// TIA Portal V18 export
FUNCTION_BLOCK "SafetyGate"   // FB5200, LAD
{ S7_Optimized_Access := 'FALSE' }
// stored: AutoNumber false, SetENOAutomatically false
   VAR_INPUT
      iSysInface : "RCS_SysComInterface_V1";
      "iSafetyGate Opened Monitor" : Bool;   // 安全门打开状态监控
      "iSafetyGate Locked Monitor" : Bool;   // 安全门锁定状态监控
      i1s_Pulse : Bool;   // 1s脉冲信号
      "iSafetyGate AutoLock Timer" : Time := T#1s;   // 安全门自动模式下锁延时
      "iSafetyGate ManualLock Timer" : Time := T#60s;   // 安全门手动模式下锁定延时
      iMode : Int;
   END_VAR
   VAR_OUTPUT
      "oSafetyGate LockedLamp" { ExternalAccessible := 'False'; ExternalVisible := 'False'; ExternalWritable := 'False'} : Bool;   // 安全门解锁输出状态
   END_VAR
   VAR_IN_OUT
      ioSafetyGateLock : Bool;   // 安全门锁定输出
      ioHMI_Interface : "SafetyGateUDT";
   END_VAR
   VAR
      "sSafetyGate Timer" { S7_SetPoint := 'True'} : Array[1..5] of TON_TIME;
      sP_Trig : Array[1..10] of Bool;
      sN_Trig : Array[1..10] of Bool;
      "sSafetyGate UnlockRequest" { ExternalAccessible := 'False'; ExternalVisible := 'False'; ExternalWritable := 'False'} : Bool;   // 安全门开门请求标志位
      "sSafetyGate LockRequest" : Bool;
   END_VAR
   VAR_TEMP
      tAlyways_On : Bool;
      tAlyways_Off : Bool;
   END_VAR
   VAR_TEMP   // added for the SCL form of the ladder/FBD networks
      _w1 : Bool;
      _w2 : Bool;
      _w3 : Bool;
      _w4 : Bool;
      _w5 : Bool;
   END_VAR
BEGIN

REGION Network 1: #tAlyways_On
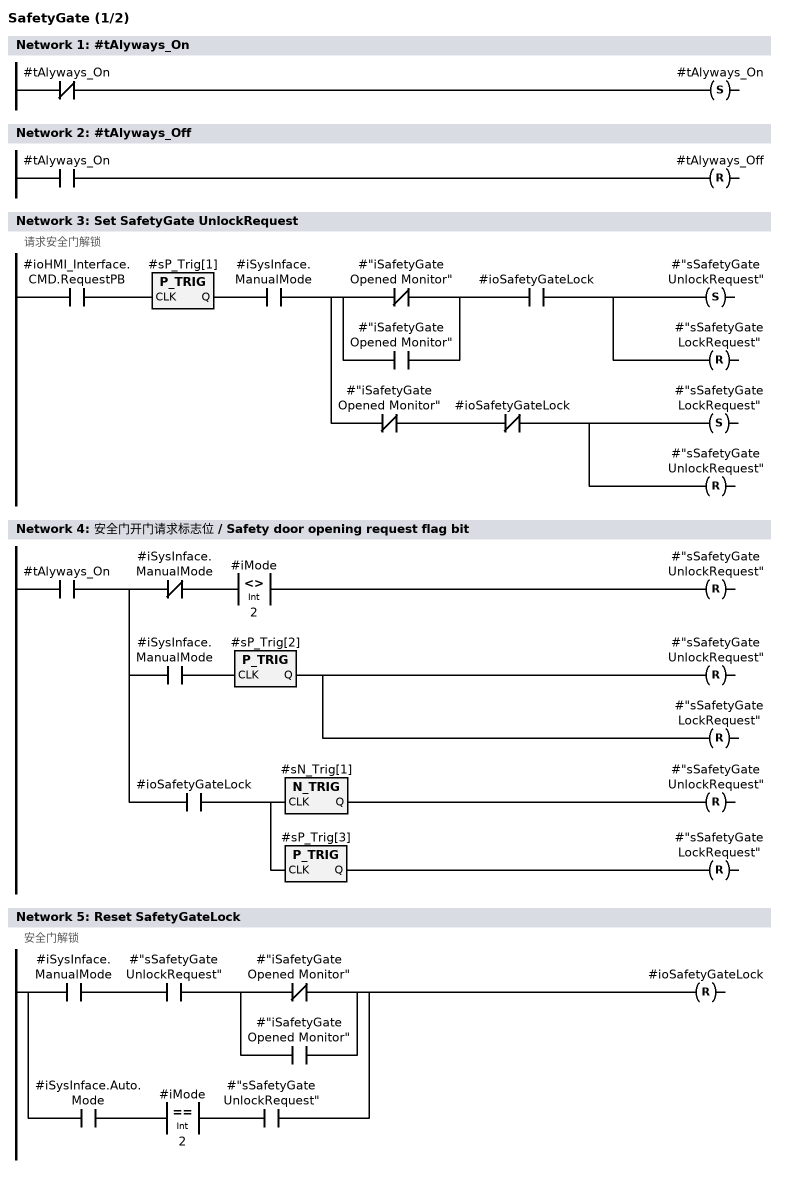
   RUNG wire#powerrail
      I_Contact( #tAlyways_On )
      S_Coil( #tAlyways_On )
   END_RUNG
   // the same network as SCL:
   IF NOT #tAlyways_On THEN #tAlyways_On := TRUE; END_IF;
END_REGION

REGION Network 2: #tAlyways_Off
   RUNG wire#powerrail
      Contact( #tAlyways_On )
      R_Coil( #tAlyways_Off )
   END_RUNG
   // the same network as SCL:
   IF #tAlyways_On THEN #tAlyways_Off := FALSE; END_IF;
END_REGION

REGION Network 3: Set SafetyGate UnlockRequest
   // 请求安全门解锁
   RUNG wire#powerrail
      Contact( #ioHMI_Interface.CMD.RequestPB )
      P_Trig( #sP_Trig[1] )
      Contact( #iSysInface.ManualMode )
      wire#w1
      I_Contact( #"iSafetyGate Opened Monitor" )
      wire#w2
      Contact( #ioSafetyGateLock )
      wire#w3
      S_Coil( #"sSafetyGate UnlockRequest" )
   END_RUNG
   RUNG wire#w1
      Contact( #"iSafetyGate Opened Monitor" )
   END_RUNG wire#w2
   RUNG wire#w3
      R_Coil( #"sSafetyGate LockRequest" )
   END_RUNG
   RUNG wire#w1
      I_Contact( #"iSafetyGate Opened Monitor" )
      I_Contact( #ioSafetyGateLock )
      wire#w4
      S_Coil( #"sSafetyGate LockRequest" )
   END_RUNG
   RUNG wire#w4
      R_Coil( #"sSafetyGate UnlockRequest" )
   END_RUNG
   // the same network as SCL:
   #_w1 := #ioHMI_Interface.CMD.RequestPB AND NOT #sP_Trig[1];   // rising edge
   #sP_Trig[1] := #ioHMI_Interface.CMD.RequestPB;
   #_w2 := #_w1 AND #iSysInface.ManualMode;
   IF #_w2 AND (NOT #"iSafetyGate Opened Monitor" OR #"iSafetyGate Opened Monitor") AND #ioSafetyGateLock THEN
       #"sSafetyGate UnlockRequest" := TRUE;
       #"sSafetyGate LockRequest" := FALSE;
   END_IF;
   IF #_w2 AND NOT #"iSafetyGate Opened Monitor" AND NOT #ioSafetyGateLock THEN
       #"sSafetyGate LockRequest" := TRUE;
       #"sSafetyGate UnlockRequest" := FALSE;
   END_IF;
END_REGION

REGION Network 4: 安全门开门请求标志位 / Safety door opening request flag bit
   RUNG wire#powerrail
      Contact( #tAlyways_On )
      wire#w1
      I_Contact( #iSysInface.ManualMode )
      { S7_Templates := "SrcType := Int" } NE_Contact(in1 := #iMode, in2 := 2)
      R_Coil( #"sSafetyGate UnlockRequest" )
   END_RUNG
   RUNG wire#w1
      Contact( #iSysInface.ManualMode )
      P_Trig( #sP_Trig[2] )
      wire#w2
      R_Coil( #"sSafetyGate UnlockRequest" )
   END_RUNG
   RUNG wire#w2
      R_Coil( #"sSafetyGate LockRequest" )
   END_RUNG
   RUNG wire#w1
      Contact( #ioSafetyGateLock )
      wire#w3
      N_Trig( #sN_Trig[1] )
      R_Coil( #"sSafetyGate UnlockRequest" )
   END_RUNG
   RUNG wire#w3
      P_Trig( #sP_Trig[3] )
      R_Coil( #"sSafetyGate LockRequest" )
   END_RUNG
   // the same network as SCL:
   IF #tAlyways_On AND NOT #iSysInface.ManualMode AND (#iMode <> 2) THEN
       #"sSafetyGate UnlockRequest" := FALSE;
   END_IF;
   #_w1 := #tAlyways_On AND #iSysInface.ManualMode;
   #_w2 := #_w1 AND NOT #sP_Trig[2];   // rising edge
   #sP_Trig[2] := #_w1;
   IF #_w2 THEN
       #"sSafetyGate UnlockRequest" := FALSE;
       #"sSafetyGate LockRequest" := FALSE;
   END_IF;
   #_w3 := #tAlyways_On AND #ioSafetyGateLock;
   #_w4 := NOT #_w3 AND #sN_Trig[1];   // falling edge
   #sN_Trig[1] := #_w3;
   IF #_w4 THEN #"sSafetyGate UnlockRequest" := FALSE; END_IF;
   #_w5 := #_w3 AND NOT #sP_Trig[3];   // rising edge
   #sP_Trig[3] := #_w3;
   IF #_w5 THEN #"sSafetyGate LockRequest" := FALSE; END_IF;
END_REGION

REGION Network 5: Reset SafetyGateLock
   // 安全门解锁
   RUNG wire#powerrail
      Contact( #iSysInface.ManualMode )
      Contact( #"sSafetyGate UnlockRequest" )
      wire#w1
      I_Contact( #"iSafetyGate Opened Monitor" )
      wire#w2
      R_Coil( #ioSafetyGateLock )
   END_RUNG
   RUNG wire#w1
      Contact( #"iSafetyGate Opened Monitor" )
   END_RUNG wire#w2
   RUNG wire#powerrail
      Contact( #iSysInface.Auto.Mode )
      { S7_Templates := "SrcType := Int" } EQ_Contact(in1 := #iMode, in2 := 2)
      Contact( #"sSafetyGate UnlockRequest" )
   END_RUNG wire#w2
   // the same network as SCL:
   IF (#iSysInface.ManualMode AND #"sSafetyGate UnlockRequest" AND (NOT #"iSafetyGate Opened Monitor" OR #"iSafetyGate Opened Monitor")) OR (#iSysInface.Auto.Mode AND (#iMode = 2) AND #"sSafetyGate UnlockRequest") THEN
       #ioSafetyGateLock := FALSE;
   END_IF;
END_REGION

REGION Network 6: Set SafetyGate Lock
   // 安全门锁定
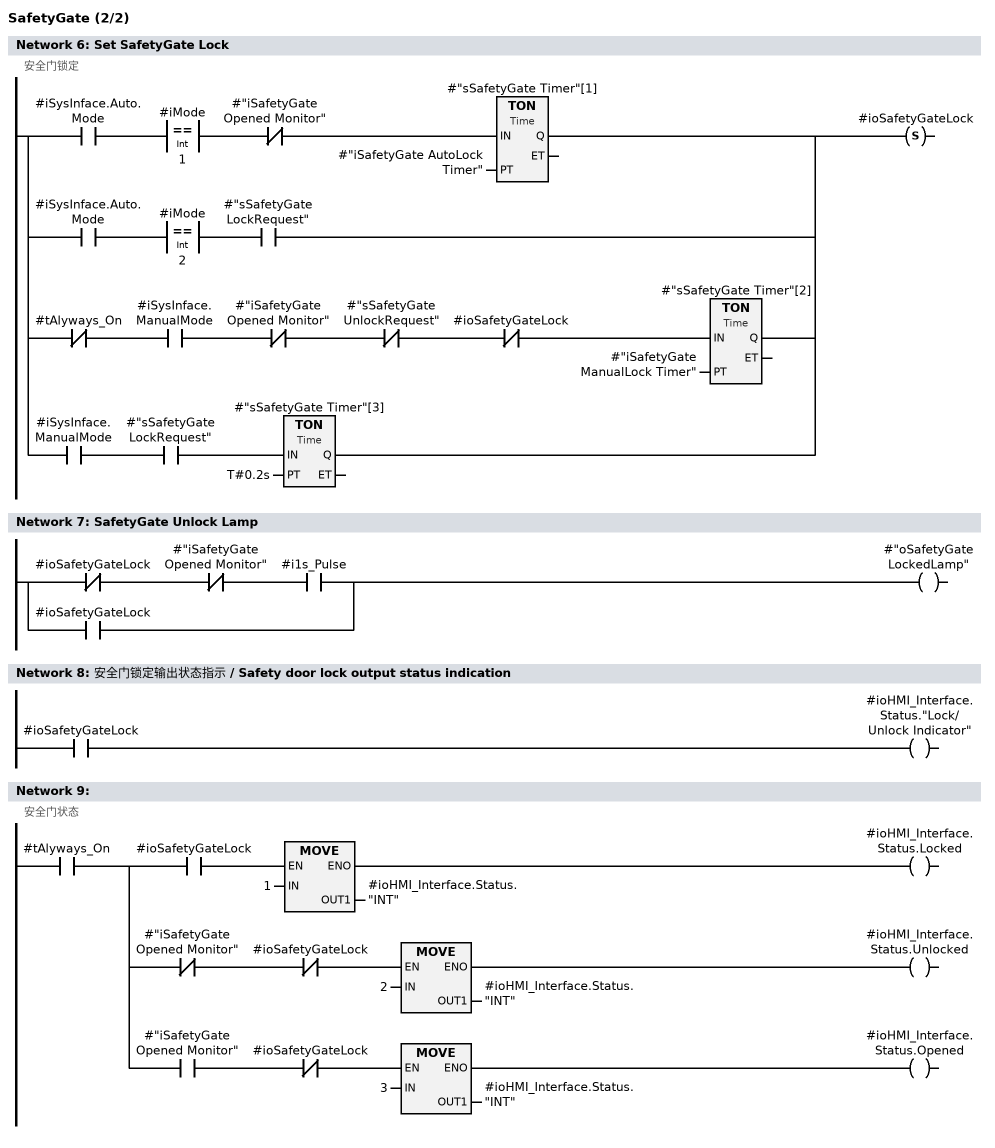
   RUNG wire#powerrail
      Contact( #iSysInface.Auto.Mode )
      { S7_Templates := "SrcType := Int" } EQ_Contact(in1 := #iMode, in2 := 1)
      I_Contact( #"iSafetyGate Opened Monitor" )
      { S7_Templates := "time_type := Time" } #"sSafetyGate Timer"[1].TON(pt := #"iSafetyGate AutoLock Timer", et =>)
      wire#w1
      S_Coil( #ioSafetyGateLock )
   END_RUNG
   RUNG wire#powerrail
      Contact( #iSysInface.Auto.Mode )
      { S7_Templates := "SrcType := Int" } EQ_Contact(in1 := #iMode, in2 := 2)
      Contact( #"sSafetyGate LockRequest" )
   END_RUNG wire#w1
   RUNG wire#powerrail
      I_Contact( #tAlyways_On )
      Contact( #iSysInface.ManualMode )
      I_Contact( #"iSafetyGate Opened Monitor" )
      I_Contact( #"sSafetyGate UnlockRequest" )
      I_Contact( #ioSafetyGateLock )
      { S7_Templates := "time_type := Time" } #"sSafetyGate Timer"[2].TON(pt := #"iSafetyGate ManualLock Timer", et =>)
   END_RUNG wire#w1
   RUNG wire#powerrail
      Contact( #iSysInface.ManualMode )
      Contact( #"sSafetyGate LockRequest" )
      { S7_Templates := "time_type := Time" } #"sSafetyGate Timer"[3].TON(pt := T#0.2s, et =>)
   END_RUNG wire#w1
   // the same network as SCL:
   #"sSafetyGate Timer"[1].TON(IN := #iSysInface.Auto.Mode AND (#iMode = 1) AND NOT #"iSafetyGate Opened Monitor",
                           PT := #"iSafetyGate AutoLock Timer");
   #_w1 := #"sSafetyGate Timer"[1].Q;
   #"sSafetyGate Timer"[2].TON(IN := NOT #tAlyways_On AND #iSysInface.ManualMode AND NOT #"iSafetyGate Opened Monitor" AND NOT #"sSafetyGate UnlockRequest" AND NOT #ioSafetyGateLock,
                           PT := #"iSafetyGate ManualLock Timer");
   #_w2 := #"sSafetyGate Timer"[2].Q;
   #"sSafetyGate Timer"[3].TON(IN := #iSysInface.ManualMode AND #"sSafetyGate LockRequest", PT := T#0.2s);
   IF #_w1 OR (#iSysInface.Auto.Mode AND (#iMode = 2) AND #"sSafetyGate LockRequest") OR #_w2 OR #"sSafetyGate Timer"[3].Q THEN
       #ioSafetyGateLock := TRUE;
   END_IF;
END_REGION

REGION Network 7: SafetyGate Unlock Lamp
   RUNG wire#powerrail
      I_Contact( #ioSafetyGateLock )
      I_Contact( #"iSafetyGate Opened Monitor" )
      Contact( #i1s_Pulse )
      wire#w1
      Coil( #"oSafetyGate LockedLamp" )
   END_RUNG
   RUNG wire#powerrail
      Contact( #ioSafetyGateLock )
   END_RUNG wire#w1
   // the same network as SCL:
   #"oSafetyGate LockedLamp" := (NOT #ioSafetyGateLock AND NOT #"iSafetyGate Opened Monitor" AND #i1s_Pulse) OR #ioSafetyGateLock;
END_REGION

REGION Network 8: 安全门锁定输出状态指示 / Safety door lock output status indication
   RUNG wire#powerrail
      Contact( #ioSafetyGateLock )
      Coil( #ioHMI_Interface.Status."Lock/Unlock Indicator" )
   END_RUNG
   // the same network as SCL:
   #ioHMI_Interface.Status."Lock/Unlock Indicator" := #ioSafetyGateLock;
END_REGION

REGION Network 9
   // 安全门状态
   RUNG wire#powerrail
      Contact( #tAlyways_On )
      wire#w1
      Contact( #ioSafetyGateLock )
      Move(in := 1, out1 => #ioHMI_Interface.Status."INT")
      Coil( #ioHMI_Interface.Status.Locked )
   END_RUNG
   RUNG wire#w1
      I_Contact( #"iSafetyGate Opened Monitor" )
      I_Contact( #ioSafetyGateLock )
      Move(in := 2, out1 => #ioHMI_Interface.Status."INT")
      Coil( #ioHMI_Interface.Status.Unlocked )
   END_RUNG
   RUNG wire#w1
      Contact( #"iSafetyGate Opened Monitor" )
      I_Contact( #ioSafetyGateLock )
      Move(in := 3, out1 => #ioHMI_Interface.Status."INT")
      Coil( #ioHMI_Interface.Status.Opened )
   END_RUNG
   // the same network as SCL:
   #_w1 := #tAlyways_On AND #ioSafetyGateLock;
   IF #_w1 THEN #ioHMI_Interface.Status."INT" := 1; END_IF;
   #ioHMI_Interface.Status.Locked := #_w1;
   #_w2 := #tAlyways_On AND NOT #"iSafetyGate Opened Monitor" AND NOT #ioSafetyGateLock;
   IF #_w2 THEN #ioHMI_Interface.Status."INT" := 2; END_IF;
   #ioHMI_Interface.Status.Unlocked := #_w2;
   #_w3 := #tAlyways_On AND #"iSafetyGate Opened Monitor" AND NOT #ioSafetyGateLock;
   IF #_w3 THEN #ioHMI_Interface.Status."INT" := 3; END_IF;
   #ioHMI_Interface.Status.Opened := #_w3;
END_REGION
END_FUNCTION_BLOCK
